{attribute addProperty BoxType "EK1100-0000-0018"}
{attribute addProperty Id "Beckhoff_EP1xxxEK1122Beckhoff_EP1xxxEK1122_A81791711312068719478376"}
{attribute addProperty CRC "1948393549"}
{attribute addProperty SizeInBites "13120"}
{attribute addProperty SizeInBytes "68719478376"}
TYPE Beckhoff_EP1xxx_7422204D EXTENDS EK1100_179A0949 :
STRUCT
	{attribute addProperty Name "Beckhoff_EP1xxxEK1122"}
	Beckhoff_EP1xxxEK1122 : Beckhoff_EP1xxxEK1122_A8179171;
END_STRUCT
END_TYPE

(* stored: Version 1.2.0.0, ProductVersion 3.1.4024.9
   DUT Beckhoff_EP1xxx_7422204D: Id {2bcac52b-70f4-4322-b0d3-75a01c9fa0f2} *)
